PROGRAM P_CloseTcHmiExe
(*program for closing the visualization (terminates Tc3PlcHMi.exe process), 
 to terminate process, set bKillProcess var to TRUE*)
VAR
	bKillProcess							: BOOL;
	ntKillProcess							: NT_StartProcess;
END_VAR

ntKillProcess(
	NETID:='' ,
	PATHSTR:='C:\WINDOWS\system32\taskkill.exe' ,
	DIRNAME:='' , 
	COMNDLINE:='/t /f /IM Tc3PlcHmi.exe' , 
	START:= bKillProcess,
	ERRID=> );
bKillProcess := FALSE;

END_PROGRAM

(* stored: Version 1.1.0.1, ProductVersion 3.1.4024.3
   POU P_CloseTcHmiExe: Id {ac59d580-afdb-42ca-8fbc-251b8ddc510f}, SpecialFunc None *)
